{attribute addProperty BoxType "EK1100-0000-0018"}
{attribute addProperty Id "Beckhoff_EL5xxxEK1122Beckhoff_EL5xxxEK1122_F18478E1162A_0001_EL5001_0000_0000EL5001_A4D8273813617A_0002_EL5001_0000_0001EL5001_A4D8273813617A_0003_EL5001_0000_1016EL5001_87A6FCF013617A_0004_EL5001_0000_1017EL5001_5BDAD4AF14418A_0005_EL5001_0000_1018EL5001_5BDAD4AF14418A_0006_EL5001_0000_1019EL5001_5BDAD4AF14418A_0007_EL5001_0000_1020EL5001_5BDAD4AF14418A_0008_EL5001_0000_1021EL5001_F220A1B714418A_0009_EL5001_0010_0000EL5001_A4D8273813617A_0010_EL5001_0011_0016EL5001_D25DCE7B24030A_0011_EL5001_0011_0017EL5001_D25DCE7B24030A_0012_EL5001_0011_0018EL5001_D25DCE7B24030A_0013_EL5001_0011_0019EL5001_E89B6F7020826A_0014_EL5001_0011_0020EL5001_E89B6F7020826A_0015_EL5001_0090_0016EL5001_636E7B5014418A_0016_EL5002_0000_0016EL5002_8CF434FD19224A_0017_EL5002_0000_0017EL5002_8CF434FD19224A_0018_EL5002_0000_0018EL5002_8CF434FD19224A_0019_EL5002_0000_0019EL5002_8CF434FD19224A_0020_EL5002_0000_0020EL5002_D767A13319224A_0021_EL5021_0000_0016EL5021_EEB77CD622428A_0022_EL5021_0000_0017EL5021_EEB77CD622428A_0023_EL5021_0000_0018EL5021_EEB77CD622428A_0024_EL5021_0000_0019EL5021_426F0F5622428A_0025_EL5021_0000_0020EL5021_426F0F5622428A_0026_EL5021_0000_0021EL5021_426F0F5622428A_0027_EL5021_0000_0022EL5021_426F0F5622428A_0028_EL5021_0090_0018EL5021_426F0F5622428A_0029_EL5021_0090_0019EL5021_426F0F5622428A_0030_EL5032_0000_0021EL5032_934FB0FD25632A_0031_EL5032_0000_0023EL5032_934FB0FD25632A_0032_EL5032_0000_0024EL5032_934FB0FD25632A_0033_EL5032_0000_0025EL5032_934FB0FD25632A_0034_EL5032_0000_0026EL5032_934FB0FD25632A_0035_EL5032_0000_0027EL5032_934FB0FD25632A_0036_EL5032_0090_0016EL5032_934FB0FD25632A_0037_EL5042_0000_0016EL5042_934FB0FD25632A_0038_EL5072_0000_0016EL5072_B22199CB36846A_0039_EL5101_0000_0000EL5101_4D0D82F516020A_0040_EL5101_0000_0001EL5101_D480A6FC16020A_0041_EL5101_0000_1017EL5101_D480A6FC16020A_0042_EL5101_0000_1018EL5101_D480A6FC16020A_0043_EL5101_0000_1019EL5101_771F729F30438A_0044_EL5101_0000_1020EL5101_3043364117622A_0045_EL5101_0000_1021EL5101_3043364117622A_0046_EL5101_0000_1022EL5101_3043364117622A_0047_EL5101_0000_1023EL5101_AD0B958A17622A_0048_EL5101_0000_1024EL5101_AD0B958A17622A_0049_EL5101_0010_0016EL5101_AF3A94C817622A_0050_EL5101_0010_0017EL5101_AF3A94C817622A_0051_EL5101_0010_0018EL5101_AF3A94C817622A_0052_EL5101_0010_0019EL5101_22B069AD17622A_0053_EL5101_0011_0016EL5101_E9B90D9532040A_0054_EL5101_0090_0016EL5101_AD0B958A17622A_0055_EL5101_0090_0017EL5101_AD0B958A17622A_0056_EL5101_1006_1019EL5101_771F729F30438A_0057_EL5101_1006_1020EL5101_3043364117622A_0058_EL5101_1006_1021EL5101_3043364117622A_0059_EL5101_1006_1022EL5101_3043364117622A_0060_EL5101_1006_1023EL5101_3043364117622A_0061_EL5151_0000_0016EL5151_0480304827234A_0062_EL5102_0000_0016EL5102_DF11825E44856A_0063_EL5112_0000_0016EL5112_0DC93E8427234A_0064_EL5122_0000_0016EL5122_C09B78AB38448A_0065_EL5151_0000_0017EL5151_AF5F3CC433642A_0066_EL5151_0000_0018EL5151_AF5F3CC433642A_0067_EL5151_0000_0019EL5151_AF5F3CC433642A_0068_EL5151_0000_0020EL5151_AFAD080A20826A_0069_EL5151_0000_0021EL5151_95571ACB20826A_0070_EL5151_0000_0022EL5151_95571ACB20826A_0071_EL5151_0000_0023EL5151_95571ACB20826A_0072_EL5151_0000_0024EL5151_95571ACB20826A_0073_EL5151_0000_0025EL5151_3376D36320826A_0074_EL5151_0000_0026EL5151_3376D36320826A_0075_EL5151_0021_0018EL5151_B58C1E4935244A_0076_EL5151_0080_0016EL5151_773FC26A28836A_0077_EL5151_0080_0017EL5151_AFAD080A20826A_0078_EL5151_0080_0018EL5151_AFAD080A20826A_0079_EL5151_0080_0019EL5151_AFAD080A20826A_0080_EL5151_0080_0020EL5151_AFAD080A20826A_0081_EL5151_0080_0021EL5151_3376D36320826A_0082_EL5151_0090_0016EL5151_867F502117622A_0083_EL5152_0000_0016EL5152_0C84728433642A_0084_EL5152_0000_0017EL5152_0C84728433642A_0085_EL5152_0000_0018EL5152_44579DF528836A_0086_EL5152_0000_0019EL5152_44579DF528836"}
{attribute addProperty CRC "1683478983"}
{attribute addProperty SizeInBites "19104"}
{attribute addProperty SizeInBytes "2388"}
TYPE Beckhoff_EL5xxx_6457D9C7 EXTENDS EK1100_179A0949 :
STRUCT
	{attribute addProperty Name "Beckhoff_EL5xxxEK1122"}
	Beckhoff_EL5xxxEK1122 : Beckhoff_EL5xxxEK1122_F18478E1;
	{attribute addProperty Name "A_0001_EL5001_0000_0000"}
	A_0001_EL5001_0000_0000 : EL5001_A4D82738;
	{attribute addProperty Name "A_0002_EL5001_0000_0001"}
	A_0002_EL5001_0000_0001 : EL5001_A4D82738;
	{attribute addProperty Name "A_0003_EL5001_0000_1016"}
	A_0003_EL5001_0000_1016 : EL5001_87A6FCF0;
	{attribute addProperty Name "A_0004_EL5001_0000_1017"}
	A_0004_EL5001_0000_1017 : EL5001_5BDAD4AF;
	{attribute addProperty Name "A_0005_EL5001_0000_1018"}
	A_0005_EL5001_0000_1018 : EL5001_5BDAD4AF;
	{attribute addProperty Name "A_0006_EL5001_0000_1019"}
	A_0006_EL5001_0000_1019 : EL5001_5BDAD4AF;
	{attribute addProperty Name "A_0007_EL5001_0000_1020"}
	A_0007_EL5001_0000_1020 : EL5001_5BDAD4AF;
	{attribute addProperty Name "A_0008_EL5001_0000_1021"}
	A_0008_EL5001_0000_1021 : EL5001_F220A1B7;
	{attribute addProperty Name "A_0009_EL5001_0010_0000"}
	A_0009_EL5001_0010_0000 : EL5001_A4D82738;
	{attribute addProperty Name "A_0010_EL5001_0011_0016"}
	A_0010_EL5001_0011_0016 : EL5001_D25DCE7B;
	{attribute addProperty Name "A_0011_EL5001_0011_0017"}
	A_0011_EL5001_0011_0017 : EL5001_D25DCE7B;
	{attribute addProperty Name "A_0012_EL5001_0011_0018"}
	A_0012_EL5001_0011_0018 : EL5001_D25DCE7B;
	{attribute addProperty Name "A_0013_EL5001_0011_0019"}
	A_0013_EL5001_0011_0019 : EL5001_E89B6F70;
	{attribute addProperty Name "A_0014_EL5001_0011_0020"}
	A_0014_EL5001_0011_0020 : EL5001_E89B6F70;
	{attribute addProperty Name "A_0015_EL5001_0090_0016"}
	A_0015_EL5001_0090_0016 : EL5001_636E7B50;
	{attribute addProperty Name "A_0016_EL5002_0000_0016"}
	A_0016_EL5002_0000_0016 : EL5002_8CF434FD;
	{attribute addProperty Name "A_0017_EL5002_0000_0017"}
	A_0017_EL5002_0000_0017 : EL5002_8CF434FD;
	{attribute addProperty Name "A_0018_EL5002_0000_0018"}
	A_0018_EL5002_0000_0018 : EL5002_8CF434FD;
	{attribute addProperty Name "A_0019_EL5002_0000_0019"}
	A_0019_EL5002_0000_0019 : EL5002_8CF434FD;
	{attribute addProperty Name "A_0020_EL5002_0000_0020"}
	A_0020_EL5002_0000_0020 : EL5002_D767A133;
	{attribute addProperty Name "A_0021_EL5021_0000_0016"}
	A_0021_EL5021_0000_0016 : EL5021_EEB77CD6;
	{attribute addProperty Name "A_0022_EL5021_0000_0017"}
	A_0022_EL5021_0000_0017 : EL5021_EEB77CD6;
	{attribute addProperty Name "A_0023_EL5021_0000_0018"}
	A_0023_EL5021_0000_0018 : EL5021_EEB77CD6;
	{attribute addProperty Name "A_0024_EL5021_0000_0019"}
	A_0024_EL5021_0000_0019 : EL5021_426F0F56;
	{attribute addProperty Name "A_0025_EL5021_0000_0020"}
	A_0025_EL5021_0000_0020 : EL5021_426F0F56;
	{attribute addProperty Name "A_0026_EL5021_0000_0021"}
	A_0026_EL5021_0000_0021 : EL5021_426F0F56;
	{attribute addProperty Name "A_0027_EL5021_0000_0022"}
	A_0027_EL5021_0000_0022 : EL5021_426F0F56;
	{attribute addProperty Name "A_0028_EL5021_0090_0018"}
	A_0028_EL5021_0090_0018 : EL5021_426F0F56;
	{attribute addProperty Name "A_0029_EL5021_0090_0019"}
	A_0029_EL5021_0090_0019 : EL5021_426F0F56;
	{attribute addProperty Name "A_0030_EL5032_0000_0021"}
	A_0030_EL5032_0000_0021 : EL5032_934FB0FD;
	{attribute addProperty Name "A_0031_EL5032_0000_0023"}
	A_0031_EL5032_0000_0023 : EL5032_934FB0FD;
	{attribute addProperty Name "A_0032_EL5032_0000_0024"}
	A_0032_EL5032_0000_0024 : EL5032_934FB0FD;
	{attribute addProperty Name "A_0033_EL5032_0000_0025"}
	A_0033_EL5032_0000_0025 : EL5032_934FB0FD;
	{attribute addProperty Name "A_0034_EL5032_0000_0026"}
	A_0034_EL5032_0000_0026 : EL5032_934FB0FD;
	{attribute addProperty Name "A_0035_EL5032_0000_0027"}
	A_0035_EL5032_0000_0027 : EL5032_934FB0FD;
	{attribute addProperty Name "A_0036_EL5032_0090_0016"}
	A_0036_EL5032_0090_0016 : EL5032_934FB0FD;
	{attribute addProperty Name "A_0037_EL5042_0000_0016"}
	A_0037_EL5042_0000_0016 : EL5042_934FB0FD;
	{attribute addProperty Name "A_0038_EL5072_0000_0016"}
	A_0038_EL5072_0000_0016 : EL5072_B22199CB;
	{attribute addProperty Name "A_0039_EL5101_0000_0000"}
	A_0039_EL5101_0000_0000 : EL5101_4D0D82F5;
	{attribute addProperty Name "A_0040_EL5101_0000_0001"}
	A_0040_EL5101_0000_0001 : EL5101_D480A6FC;
	{attribute addProperty Name "A_0041_EL5101_0000_1017"}
	A_0041_EL5101_0000_1017 : EL5101_D480A6FC;
	{attribute addProperty Name "A_0042_EL5101_0000_1018"}
	A_0042_EL5101_0000_1018 : EL5101_D480A6FC;
	{attribute addProperty Name "A_0043_EL5101_0000_1019"}
	A_0043_EL5101_0000_1019 : EL5101_771F729F;
	{attribute addProperty Name "A_0044_EL5101_0000_1020"}
	A_0044_EL5101_0000_1020 : EL5101_30433641;
	{attribute addProperty Name "A_0045_EL5101_0000_1021"}
	A_0045_EL5101_0000_1021 : EL5101_30433641;
	{attribute addProperty Name "A_0046_EL5101_0000_1022"}
	A_0046_EL5101_0000_1022 : EL5101_30433641;
	{attribute addProperty Name "A_0047_EL5101_0000_1023"}
	A_0047_EL5101_0000_1023 : EL5101_AD0B958A;
	{attribute addProperty Name "A_0048_EL5101_0000_1024"}
	A_0048_EL5101_0000_1024 : EL5101_AD0B958A;
	{attribute addProperty Name "A_0049_EL5101_0010_0016"}
	A_0049_EL5101_0010_0016 : EL5101_AF3A94C8;
	{attribute addProperty Name "A_0050_EL5101_0010_0017"}
	A_0050_EL5101_0010_0017 : EL5101_AF3A94C8;
	{attribute addProperty Name "A_0051_EL5101_0010_0018"}
	A_0051_EL5101_0010_0018 : EL5101_AF3A94C8;
	{attribute addProperty Name "A_0052_EL5101_0010_0019"}
	A_0052_EL5101_0010_0019 : EL5101_22B069AD;
	{attribute addProperty Name "A_0053_EL5101_0011_0016"}
	A_0053_EL5101_0011_0016 : EL5101_E9B90D95;
	{attribute addProperty Name "A_0054_EL5101_0090_0016"}
	A_0054_EL5101_0090_0016 : EL5101_AD0B958A;
	{attribute addProperty Name "A_0055_EL5101_0090_0017"}
	A_0055_EL5101_0090_0017 : EL5101_AD0B958A;
	{attribute addProperty Name "A_0056_EL5101_1006_1019"}
	A_0056_EL5101_1006_1019 : EL5101_771F729F;
	{attribute addProperty Name "A_0057_EL5101_1006_1020"}
	A_0057_EL5101_1006_1020 : EL5101_30433641;
	{attribute addProperty Name "A_0058_EL5101_1006_1021"}
	A_0058_EL5101_1006_1021 : EL5101_30433641;
	{attribute addProperty Name "A_0059_EL5101_1006_1022"}
	A_0059_EL5101_1006_1022 : EL5101_30433641;
	{attribute addProperty Name "A_0060_EL5101_1006_1023"}
	A_0060_EL5101_1006_1023 : EL5101_30433641;
	{attribute addProperty Name "A_0061_EL5151_0000_0016"}
	A_0061_EL5151_0000_0016 : EL5151_04803048;
	{attribute addProperty Name "A_0062_EL5102_0000_0016"}
	A_0062_EL5102_0000_0016 : EL5102_DF11825E;
	{attribute addProperty Name "A_0063_EL5112_0000_0016"}
	A_0063_EL5112_0000_0016 : EL5112_0DC93E84;
	{attribute addProperty Name "A_0064_EL5122_0000_0016"}
	A_0064_EL5122_0000_0016 : EL5122_C09B78AB;
	{attribute addProperty Name "A_0065_EL5151_0000_0017"}
	A_0065_EL5151_0000_0017 : EL5151_AF5F3CC4;
	{attribute addProperty Name "A_0066_EL5151_0000_0018"}
	A_0066_EL5151_0000_0018 : EL5151_AF5F3CC4;
	{attribute addProperty Name "A_0067_EL5151_0000_0019"}
	A_0067_EL5151_0000_0019 : EL5151_AF5F3CC4;
	{attribute addProperty Name "A_0068_EL5151_0000_0020"}
	A_0068_EL5151_0000_0020 : EL5151_AFAD080A;
	{attribute addProperty Name "A_0069_EL5151_0000_0021"}
	A_0069_EL5151_0000_0021 : EL5151_95571ACB;
	{attribute addProperty Name "A_0070_EL5151_0000_0022"}
	A_0070_EL5151_0000_0022 : EL5151_95571ACB;
	{attribute addProperty Name "A_0071_EL5151_0000_0023"}
	A_0071_EL5151_0000_0023 : EL5151_95571ACB;
	{attribute addProperty Name "A_0072_EL5151_0000_0024"}
	A_0072_EL5151_0000_0024 : EL5151_95571ACB;
	{attribute addProperty Name "A_0073_EL5151_0000_0025"}
	A_0073_EL5151_0000_0025 : EL5151_3376D363;
	{attribute addProperty Name "A_0074_EL5151_0000_0026"}
	A_0074_EL5151_0000_0026 : EL5151_3376D363;
	{attribute addProperty Name "A_0075_EL5151_0021_0018"}
	A_0075_EL5151_0021_0018 : EL5151_B58C1E49;
	{attribute addProperty Name "A_0076_EL5151_0080_0016"}
	A_0076_EL5151_0080_0016 : EL5151_773FC26A;
	{attribute addProperty Name "A_0077_EL5151_0080_0017"}
	A_0077_EL5151_0080_0017 : EL5151_AFAD080A;
	{attribute addProperty Name "A_0078_EL5151_0080_0018"}
	A_0078_EL5151_0080_0018 : EL5151_AFAD080A;
	{attribute addProperty Name "A_0079_EL5151_0080_0019"}
	A_0079_EL5151_0080_0019 : EL5151_AFAD080A;
	{attribute addProperty Name "A_0080_EL5151_0080_0020"}
	A_0080_EL5151_0080_0020 : EL5151_AFAD080A;
	{attribute addProperty Name "A_0081_EL5151_0080_0021"}
	A_0081_EL5151_0080_0021 : EL5151_3376D363;
	{attribute addProperty Name "A_0082_EL5151_0090_0016"}
	A_0082_EL5151_0090_0016 : EL5151_867F5021;
	{attribute addProperty Name "A_0083_EL5152_0000_0016"}
	A_0083_EL5152_0000_0016 : EL5152_0C847284;
	{attribute addProperty Name "A_0084_EL5152_0000_0017"}
	A_0084_EL5152_0000_0017 : EL5152_0C847284;
	{attribute addProperty Name "A_0085_EL5152_0000_0018"}
	A_0085_EL5152_0000_0018 : EL5152_44579DF5;
	{attribute addProperty Name "A_0086_EL5152_0000_0019"}
	A_0086_EL5152_0000_0019 : EL5152_44579DF5;
END_STRUCT
END_TYPE

(* stored: Version 1.2.0.0, ProductVersion 3.1.4024.9
   DUT Beckhoff_EL5xxx_6457D9C7: Id {09d6f746-f34c-47d4-9faa-ce0f36435e59} *)
